TYPE chillerType :
(
	ChillerType_Default := 0, //常规水冷机
	ChillerType_Vacuum := 1, // 未知1
	ChillerType_ButV := 2 // 未知1
)UINT;
END_TYPE

(* stored: Version 1.1.0.1, ProductVersion 3.1.4024.4
   DUT chillerType: Id {a0131947-e3d5-41d5-b369-80ab83c6e895} *)
